// TIA Portal V20 export
DATA_BLOCK "ProdDataInterfaceHmi"   // DB53
TITLE = HMI und Anwender Schnittstelle für Produktionsdaten / HMI and user interface for production data
AUTHOR : SICAR
FAMILY : ProdData
// FUNKTIONSBESCHREIBUNG: 
// Der Baustein beinhaltet alle Informationen zum und vom HMI, sowie die Anwenderschnittstellen für die Produktionsdaten
// Weitere Hinweise: siehe SICAR anwenderdefinierte Dokumentation / SICAR Online-Hilfe.
// DESCRIPTION OF FUNCTIONS:
// stored: MemoryReserve 100
   VAR RETAIN
      numberOfDataSets : "LSicar_typeNumberOfDataSets";   // Anzahl konfigurierter Datensätze / Number of configured data sets
   END_VAR
   VAR
      colorCodeLimitSummary : UInt;   // Gesamt Status Grenzwerte / Overall status Limit values
      colorCodeLimitSelButton : Array[0..8] of UInt;   // Farbcode für Datensatz Anwahl Button (Grenzwerte) / Color code for data set select button (Limit values)
   END_VAR
   VAR RETAIN
      counterDataSetSel : Int := 1;   // Angewählter Datensatz Zaehler / selected data set counter
      counterDataSet : Array[0.."NO_DATASETS_COUNTER"] of "LSicar_typeCounter";   // Datensätze Zähler / Data sets counter
      cycleTimerDataSetSel : Int := 1;   // Angewaehlter Datensatz Taktzeiten / selected data set cycle timer
      cycleTimerDataSet : Array[0.."NO_DATASETS_CYCLETIMER"] of "LSicar_typeCycleTimer";   // Datensätze Taktzeiten / Data sets cycle timer
      limitValueDataSetSel : Int := 1;   // Angwaehlter Datensatz Grenzwerte / selected data set limit values
      limitDataSet : Array[0.."NO_DATASETS_LIMITVALUES"] of "LSicar_typeLimitValue";   // Datensätze Grenzwerte / Data sets limit .values
      shiftCounterDataSetSel : Int := 1;   // Angewaehlter Datensatz Schichtzaehler / selected data set shift counter
      shiftCounterDataSet : Array[0.."NO_DATASETS_SHIFTCOUNTER"] of "LSicar_typeShiftCounter";   // Datensätze Schichtzähler / Data sets shift counter
      shiftCountOeeDataSetSel : Int := 1;   // Angewaehlter Datensatz OEE / selected data set OEE
      shiftCounterOeeDataSet : Array[0.."NO_DATASETS_SHIFTCOUNTER"] of "LSicar_typeShiftCounterOee";   // Datensätze Schichtzähler OEE / Data sets shift counter OEE
   END_VAR
BEGIN
END_DATA_BLOCK
